// TIA Portal V19 export
DATA_BLOCK "SpProd"   // DB220
{ S7_Optimized_Access := 'TRUE' }
AUTHOR : CH
FAMILY : Aktina
NAME : SEQUENCE
// stored: AutoNumber false, MemoryReserve 100
   VAR RETAIN
      drill { S7_SetPoint := 'True'} : "dtDrill";
      supply : "dtSupply";
   END_VAR
   VAR
      iTank { S7_SetPoint := 'True'} : Array[0..1] of "UDT_TANKPRESS_2";
      autoReset { S7_SetPoint := 'True'} : Array[0..0] of "dtAutoReset";
   END_VAR
BEGIN
   drill.level[0] := 75;
   drill.level[1] := 85;
   drill.level[2] := 90;
   drill.level[3] := 100;
   drill.tDelay := T#5S;
   drill.setPriority[0] := 2;
   drill.setPriority[1] := 3;
   drill.setPriority[2] := 0;
   drill.loadPriority[0] := 2;
   drill.loadPriority[1] := 3;
   drill.loadPriority[2] := 0;
   drill.TankAvailable[0..1] := TRUE;
   drill.loadBtn := FALSE;
   supply.setAvailPumps[0] := FALSE;
   supply.setAvailPumps[1..3] := TRUE;
   supply.loadAvailPumps[0] := FALSE;
   supply.loadAvailPumps[1..3] := TRUE;
   supply.availPumps[0..2] := TRUE;
   supply.loadBtn := FALSE;
   supply.pressureSP := 4.0;
   supply.hhPressureAlm := 6.0;
   supply.highFlow := 35.0;
   supply.lowFlow := 10.0;
   supply.zChangeThr := 0.3;
   supply.zChangeDelay := T#1S;
   supply.PumpInterval := T#10H;
   supply.zoneChangeOP := 90.0;
   supply.overlapDelay := T#10S;
   supply.downgradeDelay := T#40S;
   supply.chLead := 2;
   supply.enRotation := FALSE;
   supply.stageUp.zoneChangeOP := 95.0;
   supply.stageUp.delayUpgrade := T#5S;
   // supply.stageDown[0] : bigPump
   // supply.stageDown[1] : midPump
   // supply.stageDown[2] : smallPump
   supply.stageDown[0..3].zoneChangeOP := 40.0;
   supply.stageDown[0..3].prevOP := 20.0;
   supply.stageDown[0..3].nextOP := 70.0;
   supply.stageDown[0].stabilizeDelay := T#1M;
   supply.stageDown[1].stabilizeDelay := T#10S;
   supply.stageDown[2..3].stabilizeDelay := T#5S;
   supply.stageDown[0..3].followUp := FALSE;
   iTank[0..1].r := 1.0;
   iTank[0..1].d := 263.0;
   iTank[0..1].hPt := 0.0;
   iTank[0..1].hBase := 0.0;
   iTank[0..1].hCyl := 525.0;
   iTank[0].hAct := 465.6394;
   iTank[1].hAct := 463.0353;
   iTank[0].vol := 25295.94;
   iTank[1].vol := 25154.47;
   // autoReset[0] : Grid
   autoReset[0].maxAlarms := 10;
   autoReset[0].perT := T#1H;
   autoReset[0].autoresetT := T#30S;
END_DATA_BLOCK
